# EPICS StreamDevice protocol: ip/ipApp/Db/SR830.proto
Terminator = CR;
extraInput=ignore;
snap {
   out "SNAP?1,2,3,4,9";
   in "%(\$1:X.VAL)f,%(\$1:Y.VAL)f,%(\$1:R.VAL)f,%(\$1:TH.VAL)f,%(\$1:REF.VAL)f";
}
